{attribute 'qualified_only'}
{attribute 'strict'}
{attribute 'to_string'}
TYPE Box_Phase :
(
	Start, Run, Delay, PushFall, PushRise, TargetCheck, Clamp, Drop, Hold 
);
END_TYPE

(* stored: Version 1.1.0.1
   DUT Box_Phase: Id {bb5b7292-25dd-4dda-9289-ce5019d6c8b8} *)
